PROGRAM MAIN
VAR
END_VAR

END_PROGRAM

(* stored: Version 1.1.0.1
   POU MAIN: Id {6b108866-eefc-481e-bf07-dfe2e0cd9452} *)
